# B&R Automation Studio project Task_1
Automation Studio 4.9

## Logical view

Binary libraries used (declarations not repeated): operator, runtime, astime, AsIecCon, Acp10man, Acp10par, NcGlobal, Acp10_MC, sys_lib, brsystem, Acp10sim, MpAxis, MpCom, MpBase, AsTCP, standard, AsArLog, AsBrStr

### Global.var - Global variables
```iecst
VAR RETAIN
	MyGlobal : {REDUND_UNREPLICABLE} UDINT := 10;
END_VAR
VAR
	gAxis01 : ACP10AXIS_typ;
	gAxis02 : ACP10AXIS_typ;
	START_BUTTON : BOOL;
	TRIGGER_INPUT : BOOL;
	EMERGENCY_STOP : BOOL;
	GreenLight : BOOL;
	RedLight : BOOL;
	CutterPosition : LREAL;
	ConveyorPosition : LREAL;
	STOP : BOOL;
	CONVEYOR_SPEED : {REDUND_UNREPLICABLE} INT := 0;
	EmergencyLight : BOOL;
	ERROR_RESET : BOOL;
	RealConveyorSpeed : INT;
	REG_TRIGGER : BOOL;
	CUTTER_POSITION : INT;
END_VAR
```

### Package Logical/Libraries - Global libraries

### Library Logical/Libraries/MyLib (IEC)

#### Types.typ - Exported data types
```iecst
TYPE
	GA_State :
		(
		NotPowered,
		WaitPower,
		Powered,
		CheckCommand,
		MoveVelocity,
		CheckVelocity,
		MoveAdditive,
		AxisHalt,
		AxisStop
		);
	COMMANDS :
		(
		NONE,
		MOVE_VELOCITY,
		MOVE_ADDITIVE,
		AXIS_HALT,
		AXIS_STOP
		);
END_TYPE
```

#### Constants.var - Exported constants
```iecst
VAR CONSTANT
	STANDSTILL : WORD := 2#00001000;
	DISCRETE_MOTION : WORD := 2#00010000;
	CONTINUOUS_MOTION : WORD := 2#00100000;
	CUTTER_SPEED : REAL := 200.0;
	CUTTER_END_POSE : REAL := 50.0;
	BELT_DISTANCE : REAL := 100.0;
END_VAR
```

#### MyLib.fun - Exported functions and function blocks
```iecst
FUNCTION_BLOCK GenericAxis_FB (*$GROUP=User,$CAT=User,$GROUPICON=User.png,$CATICON=User.png*)
	VAR_INPUT
		AxisOperation : INT;
		AxisCommand : COMMANDS;
		Master : UDINT;
		Slave : UDINT;
		CamTable : STRING[12];
		Position : REAL;
		Velocity : REAL;
		Acceleration : REAL;
		Deceleration : REAL;
		Jerk : REAL;
		Direction : USINT;
		ArraySize : INT;
		Scale : REAL;
		Offset : REAL;
		RatioNumerator : INT;
		RatioDenominator : INT;
	END_VAR
	VAR_OUTPUT
		CommandExecuted : BOOL;
		CommandAborted : BOOL;
		Error : BOOL;
		ErrorID : UINT;
		AxisErrorID : UINT;
		AxisErrorCount : UINT;
		AxisNotInitialized : BOOL;
		Status : WORD;
		ActualVelocity : REAL;
		ActualPosition : LREAL;
	END_VAR
	VAR_IN_OUT
		AxisEnable : BOOL;
	END_VAR
	VAR
		OldVelocity : REAL;
		MC_Power_GA : MC_Power;
		MC_Home_GA : MC_Home;
		MC_MoveVelocity_GA : MC_MoveVelocity;
		MC_MoveAdditive_GA : MC_MoveAdditive;
		MC_MoveAbsolute_GA : MC_MoveAbsolute;
		MC_ReadActualPosition_GA : MC_ReadActualPosition;
		MC_ReadActualVelocity_GA : MC_ReadActualVelocity;
		MC_ReadAxisError_GA : MC_ReadAxisError;
		MC_ReadStatus_GA : MC_ReadStatus;
		AxisState : GA_State;
		MC_Halt_GA : MC_Halt;
		MC_Stop_GA : MC_Stop;
	END_VAR
END_FUNCTION_BLOCK
```

#### GenericAxis_FB.st
```iecst
FUNCTION_BLOCK GenericAxis_FB
	CASE (AxisState) OF
		NotPowered:
			IF AxisEnable THEN
				MC_Power_GA.Enable := TRUE;
				AxisState := WaitPower;
			END_IF;
		WaitPower:
			IF MC_Power_GA.Status THEN
				MC_Home_GA.Execute := TRUE;
				AxisState := Powered;
			END_IF;
		Powered:
			IF MC_Home_GA.Done THEN
				MC_Home_GA.Execute := FALSE;
				AxisEnable := FALSE;
				CommandExecuted := TRUE;
				AxisState := CheckCommand; //ready state in the prof's slides
			END_IF
		// In this state you can implement several commands
		CheckCommand:
			IF AxisCommand = MOVE_VELOCITY THEN
				CommandExecuted := FALSE;
				MC_MoveVelocity_GA.Execute := TRUE;
				AxisState := MoveVelocity;
			END_IF

			IF AxisCommand = MOVE_ADDITIVE THEN
				CommandExecuted := FALSE;
				MC_MoveAdditive_GA.Execute := TRUE;
				AxisState := MoveAdditive;
			END_IF

			IF AxisCommand = AXIS_HALT THEN
				CommandExecuted := FALSE;
				MC_Halt_GA.Execute := TRUE;
				AxisState := AxisHalt;
			END_IF

			IF AxisCommand = AXIS_STOP THEN
				CommandExecuted := FALSE;
				MC_Stop_GA.Execute := TRUE;
				AxisState := AxisStop;
			END_IF

			(*IF AxisCommand = NONE THEN
				CommandExecuted := FALSE;
			END_IF*)

		// command states
		MoveVelocity:
			IF MC_MoveVelocity_GA.InVelocity THEN
				CommandExecuted := TRUE;
				MC_MoveVelocity_GA.Execute := FALSE;
				AxisState := CheckVelocity;
			END_IF
			IF (AxisCommand <> MOVE_VELOCITY) THEN
				CommandExecuted := FALSE;
				AxisState := CheckCommand;
			END_IF
		CheckVelocity:
			IF (Velocity <> OldVelocity) THEN
				OldVelocity := Velocity;
				MC_MoveVelocity_GA.Execute := TRUE;
				AxisState := MoveVelocity;
			END_IF
			IF (AxisCommand <> MOVE_VELOCITY) THEN
				CommandExecuted := FALSE;
				AxisState := CheckCommand;

			END_IF

		MoveAdditive:
			IF MC_MoveAdditive_GA.Done THEN
				MC_MoveAdditive_GA.Execute := FALSE;
				AxisCommand := NONE;
				AxisState := CheckCommand;
				CommandExecuted := TRUE;
			ELSIF (AxisCommand <> MOVE_ADDITIVE) THEN
				MC_MoveAdditive_GA.Execute := FALSE;
				CommandExecuted := FALSE;
				AxisState := CheckCommand;

			END_IF

			// In my implementation I used Halt to stop in Emergency conditions. IT IS NOT CORRECT
			// TO DO: Implement Halt in normal conditions and use STOP for critical conditions
		AxisHalt:
			IF MC_Halt_GA.Done THEN
				CommandExecuted := TRUE;
				MC_Halt_GA.Execute := FALSE;
				AxisState := NotPowered; // It goes to the NotPowered state to perform a full reset of the system
				MC_Power_GA.Enable := FALSE; // The power is disabled for the same reason
				AxisCommand := NONE;
			END_IF

		// TO DO: IT IS NOT IMPLEMENTED  (To stop the execution in critical conditions)
		AxisStop:
			IF MC_Stop_GA.Done THEN
				CommandExecuted := TRUE;
				MC_Stop_GA.Execute := FALSE;
				AxisState := NotPowered; // It goes to the NotPowered state to perform a full reset of the system
				MC_Power_GA.Enable := FALSE; // The power is disabled for the same reason
				AxisCommand := NONE;
			END_IF
	END_CASE;

	MC_Power_GA.Axis := Slave;
	MC_Power_GA();
	MC_Home_GA.Axis := Slave;
	MC_Home_GA.Position := 0;
	MC_Home_GA();
	MC_MoveVelocity_GA.Axis := Slave;
	MC_MoveVelocity_GA.Velocity := Velocity;
	MC_MoveVelocity_GA.Acceleration := Acceleration;
	MC_MoveVelocity_GA.Deceleration := Deceleration;
	MC_MoveVelocity_GA();

	MC_MoveAdditive_GA.Axis := Slave;
	MC_MoveAdditive_GA.Distance := Position;
	MC_MoveAdditive_GA.Velocity := Velocity;
	MC_MoveAdditive_GA.Acceleration := Acceleration;
	MC_MoveAdditive_GA.Deceleration := Deceleration;
	MC_MoveAdditive_GA();

	// Stop in normal conditions
	MC_Halt_GA.Axis := Slave;
	MC_Halt_GA.Deceleration := Deceleration;
	MC_Halt_GA();

	// Stop in critical conditions
	MC_Stop_GA.Axis := Slave;
	MC_Stop_GA.Deceleration := Deceleration;
	MC_Stop_GA();

	// FEEDBACKS
	MC_ReadActualPosition_GA.Axis := Slave;
	MC_ReadActualPosition_GA.Enable := TRUE;
	MC_ReadActualPosition_GA();
	ActualPosition := MC_ReadActualPosition_GA.Position;
	MC_ReadActualVelocity_GA.Axis := Slave;
	MC_ReadActualVelocity_GA.Enable := TRUE;
	MC_ReadActualVelocity_GA();
	ActualVelocity := MC_ReadActualVelocity_GA.Velocity;
	MC_ReadAxisError_GA.Enable := TRUE;
	MC_ReadAxisError_GA.Axis := Slave;
	MC_ReadAxisError_GA();
	Error := MC_ReadAxisError_GA.Error;
	ErrorID := MC_ReadAxisError_GA.ErrorID;
	AxisErrorID := MC_ReadAxisError_GA.AxisErrorID;
	AxisErrorCount := MC_ReadAxisError_GA.AxisErrorCount;
	MC_ReadStatus_GA.Enable := TRUE;
	MC_ReadStatus_GA.Axis := Slave;
	MC_ReadStatus_GA();

	IF MC_ReadStatus_GA.ContinuousMotion THEN
		Status := CONTINUOUS_MOTION;
	END_IF
	IF MC_ReadStatus_GA.DiscreteMotion THEN
		Status := DISCRETE_MOTION;
	END_IF
	IF MC_ReadStatus_GA.StandStill THEN
		Status := STANDSTILL;
	END_IF
END_FUNCTION_BLOCK
```

### Library Logical/Libraries/ComTCP/ComTCP_L (ANSIC)

#### MNG_CpyMsgToInp.cpp
```cpp
#include "MNG_InternalTyp.hpp"

unsigned long int MNG_CpyMsgToInp(MNG_RawDatagram * pFromServer, ComTCP_INPUTS_32BIT_FWRD *pSimInputs) {

    MNG_DatagramType datagramType;
	unsigned long int DWordBuffer;
        unsigned long int byteCount;
	unsigned long int numSignalsInMessage;

	byteCount = N_TO_HUDINT((pFromServer->Header).ByteCount);
	datagramType = static_cast<MNG_DatagramType>(N_TO_HUDINT((pFromServer->Header).DatagramType));
	if (datagramType != MNG_Raw32BitImage) {
		return 0;
	}

    pSimInputs->NumSignals = 15;

    numSignalsInMessage = N_TO_HUDINT(pFromServer->Payload[0]);
        if ((static_cast<long int>(numSignalsInMessage) != pSimInputs->NumSignals) ||
	(byteCount != 4 + numSignalsInMessage * 4)) {
		return 0;
	}

    /* BOOL Emergency_Button_ButtonToggle */
    pSimInputs->Emergency_Button_ButtonToggle = (pFromServer->Payload[1] != 0);

    /* BOOL Yellow_Button_ButtonPress */
    pSimInputs->Yellow_Button_ButtonPress = (pFromServer->Payload[2] != 0);

    /* BOOL White_Button_ButtonPress */
    pSimInputs->White_Button_ButtonPress = (pFromServer->Payload[3] != 0);

    /* BOOL Start_Button_ButtonPress */
    pSimInputs->Start_Button_ButtonPress = (pFromServer->Payload[4] != 0);

    /* BOOL Stop_Button_ButtonPress */
    pSimInputs->Stop_Button_ButtonPress = (pFromServer->Payload[5] != 0);

    /* FLOAT32 Knob_0_AXIS */
    DWordBuffer = N_TO_HUDINT(pFromServer->Payload[6]);
    brsmemcpy((unsigned long int)&(pSimInputs->Knob_0_AXIS), (unsigned long int)&(DWordBuffer), 4);

    /* FLOAT32 Knob_1_AXIS */
    DWordBuffer = N_TO_HUDINT(pFromServer->Payload[7]);
    brsmemcpy((unsigned long int)&(pSimInputs->Knob_1_AXIS), (unsigned long int)&(DWordBuffer), 4);

    /* FLOAT32 Knob_2_AXIS */
    DWordBuffer = N_TO_HUDINT(pFromServer->Payload[8]);
    brsmemcpy((unsigned long int)&(pSimInputs->Knob_2_AXIS), (unsigned long int)&(DWordBuffer), 4);

    /* FLOAT32 Knob_3_AXIS */
    DWordBuffer = N_TO_HUDINT(pFromServer->Payload[9]);
    brsmemcpy((unsigned long int)&(pSimInputs->Knob_3_AXIS), (unsigned long int)&(DWordBuffer), 4);

    /* FLOAT32 Shaft_1_AXIS */
    DWordBuffer = N_TO_HUDINT(pFromServer->Payload[10]);
    brsmemcpy((unsigned long int)&(pSimInputs->Shaft_1_AXIS), (unsigned long int)&(DWordBuffer), 4);

    /* BOOL Shaft_1_LBK */
    pSimInputs->Shaft_1_LBK = (pFromServer->Payload[11] != 0);

    /* BOOL Shaft_1_LFR */
    pSimInputs->Shaft_1_LFR = (pFromServer->Payload[12] != 0);

    /* FLOAT32 Shaft_0_AXIS */
    DWordBuffer = N_TO_HUDINT(pFromServer->Payload[13]);
    brsmemcpy((unsigned long int)&(pSimInputs->Shaft_0_AXIS), (unsigned long int)&(DWordBuffer), 4);

    /* BOOL Shaft_0_LBK */
    pSimInputs->Shaft_0_LBK = (pFromServer->Payload[14] != 0);

    /* BOOL Shaft_0_LFR */
    pSimInputs->Shaft_0_LFR = (pFromServer->Payload[15] != 0);

return N_TO_HUDINT((pFromServer->Header).Counter); // return counter
}
```

#### MNG_CpyOutToMsg.cpp
```cpp
#include "MNG_InternalTyp.hpp"

unsigned long int MNG_CpyOutToMsg(MNG_RawDatagram * pToServer, unsigned long int counter, ComTCP_OUTPUTS_32BIT_FWRD *pSimOutputs ) {

        unsigned long int DWordBuffer;

        pSimOutputs->NumSignals = 6;
        (pToServer->Header).ByteCount    = H_TO_NUDINT(28);
        (pToServer->Header).DatagramType = H_TO_NUDINT(MNG_Raw32BitImage);
        (pToServer->Header).SentTime = H_TO_NUDINT(0);  // Todo
        (pToServer->Header).Counter = H_TO_NUDINT(counter);
        pToServer->Payload[0] = H_TO_NUDINT(pSimOutputs->NumSignals);

    /* Yellow_light_Key : UINT32 */
    pToServer->Payload[1] = H_TO_NUDINT(pSimOutputs->Yellow_light_Key);

    /* Stop_light_Key : UINT32 */
    pToServer->Payload[2] = H_TO_NUDINT(pSimOutputs->Stop_light_Key);

    /* White_light_Key : UINT32 */
    pToServer->Payload[3] = H_TO_NUDINT(pSimOutputs->White_light_Key);

    /* Green_light_Key : UINT32 */
    pToServer->Payload[4] = H_TO_NUDINT(pSimOutputs->Green_light_Key);

    /* Shaft_0_ACT_POS : FLOAT32 */
    brsmemcpy((unsigned long int)&(DWordBuffer), (unsigned long int)&(pSimOutputs->Shaft_0_ACT_POS), 4);
    pToServer->Payload[5] = H_TO_NUDINT(DWordBuffer);

    /* Shaft_1_ACT_POS : FLOAT32 */
    brsmemcpy((unsigned long int)&(DWordBuffer), (unsigned long int)&(pSimOutputs->Shaft_1_ACT_POS), 4);
    pToServer->Payload[6] = H_TO_NUDINT(DWordBuffer);

	return 0;
}
```

### Package Logical/gAxis01obj - gAxis01obj

### gAxis01i.ax
```
InitParameter (Version=5.24.1, NcSwId=ACP10)
  ACP10AXIS_typ:
    dig_in:
      level:
        reference = ncACTIV_HI
        pos_hw_end = ncACTIV_HI
        neg_hw_end = ncACTIV_HI
        trigger1 = ncACTIV_HI
        trigger2 = ncACTIV_HI
    encoder_if:
      parameter:
        count_dir = ncSTANDARD
        scaling:
          load:
            units = 360
            rev_motor = 1
    limit:
      parameter:
        v_pos = 10000.0
        v_neg = 10000.0
        a1_pos = 50000.0
        a2_pos = 50000.0
        a1_neg = 50000.0
        a2_neg = 50000.0
        t_jolt = 0.0
        t_in_pos = 0.0
        pos_sw_end = 2000000000
        neg_sw_end = -2000000000
        ds_warning = 500.0
        ds_stop = 1000.0
        a_stop = 1.0E+30
        dv_stop = 0.0
        dv_stop_mode = ncOFF
    controller:
      mode = ncPOSITION
      position:
        kv = 349.0
        tn = 0.0
        t_predict = 0.0004
        t_total = 0.0004
        p_max = 1.0E+30
        i_max = 0.0
      speed:
        kv = 0.65
        tn = 0.0
        t_filter = 0.0
        isq_filter1:
          type = ncOFF
          a0 = 0.0
          a1 = 0.0
          b0 = 0.0
          b1 = 0.0
          b2 = 0.0
          c0_par_id = 0
          c1_par_id = 0
        isq_filter2:
          type = ncOFF
          a0 = 0.0
          a1 = 0.0
          b0 = 0.0
          b1 = 0.0
          b2 = 0.0
          c0_par_id = 0
          c1_par_id = 0
        isq_filter3:
          type = ncOFF
          a0 = 0.0
          a1 = 0.0
          b0 = 0.0
          b1 = 0.0
          b2 = 0.0
          c0_par_id = 0
          c1_par_id = 0
      uf:
        type = ncLINEAR + ncCORRECTION
        auto_config = ncMOTOR_PAR
        u0 = 0.0
        un = 0.0
        fn = 50.0
        k_f_slip = 0.0
      ff:
        mode = ncSTANDARD
        torque_load = 0.0
        torque_pos = 0.0
        torque_neg = 0.0
        kv_torque = 0.0
        inertia = 0.0
        t_filter_a = 0.0
      fb:
        mode = ncSTANDARD
        speed_mix_ratio = 0.0
        speed_kv = 0.0
      model:
        mass1:
          inertia = 0.0
          viscous_friction = 0.0
        mass2:
          inertia = 0.0
          viscous_friction = 0.0
          stiffness = 0.0
          damping = 0.0
    move:
      stop:
        parameter[0]:
          decel_ramp = ncA_LIMIT
          controller = ncON
        parameter[1]:
          decel_ramp = ncA_LIMIT
          controller = ncON
        parameter[2]:
          decel_ramp = ncA_LIMIT
          controller = ncON
        parameter[3]:
          decel_ramp = ncA_LIMIT
          controller = ncON
        quickstop:
          decel_ramp = ncA_LIMIT
          t_jolt = 0.0
        drive_error:
          decel_ramp = ncA_LIMIT
      homing:
        parameter:
          s = 0
          v_switch = 5000.0
          v_trigger = 500.0
          a = 50000.0
          mode = ncDIRECT
          edge_sw = ncPOSITIVE
          start_dir = ncPOSITIVE
          trigg_dir = ncPOSITIVE
          ref_pulse = ncOFF
          fix_dir = ncOFF
          tr_s_block = 0.0
          torque_lim = 0.0
          ds_block = 0.0
          ds_stop = 0.0
      basis:
        parameter:
          v_pos = 360.0
          v_neg = 5000.0
          a1_pos = 50000.0
          a2_pos = 50000.0
          a1_neg = 50000.0
          a2_neg = 50000.0
    message:
      text:
        parameter:
          format = ncBREAK
          columns = 80
          data_modul = acp10etxen
```

### Program Logical/PROGRAM1 (IEC)

#### Types.typ
```iecst
TYPE
	State_type :
		(
		CutterMoveBackward,
		CutterCompleted,
		CutterMoveForward,
		ConveyorStopping,
		ConveyorMoving,
		ConveyorStarting,
		AxisEnabled,
		InitializeAxis,
		CutterBackward,
		CutterForward,
		ConveyorHolding,
		WaitProduct,
		Initialize,
		Init,
		StopState,
		HaltState,
		WaitForConveyor,
		CheckReset,
		RegulatePosition
		);
END_TYPE
```

#### Variables.var
```iecst
VAR
	MachineState : State_type;
	ConveyorEnable : BOOL;
	CutterEnable : BOOL;
	Cutter : GenericAxis_FB;
	Conveyor : GenericAxis_FB;
	InitializeConveyor : BOOL;
	InitializeCutter : BOOL;
	ConveyorDisable : BOOL;
	CutterDisable : BOOL;
	ConveyorState : State_type;
	CutterState : State_type;
	ConveyorAxisEnable : BOOL;
	CutterAxisEnable : BOOL;
	FutureStop : BOOL;
	CoveyorState : BOOL;
	ConveyorStopped : BOOL;
	CutterStopped : BOOL;
	EmergencyStateMachine : INT;
	Count : INT;
	ToggleLights : BOOL;
	OldCutterPose : INT;
END_VAR
```

#### Main.st
```iecst
PROGRAM _INIT
	(* Insert code here *)
	MachineState := Init;
	ConveyorState := Init;
	CutterState := Init;
	OldCutterPose := 0;
END_PROGRAM

PROGRAM _CYCLIC

	// STOP indicates an emergency stop, it is not a stop in normal conditions
	CASE EmergencyStateMachine OF
		0 :
			IF EMERGENCY_STOP THEN
				MachineState := StopState;
				ConveyorState := StopState;
				CutterState := StopState;
				Conveyor.AxisCommand := AXIS_HALT;
				Cutter.AxisCommand := AXIS_HALT;
				EmergencyStateMachine := 1;
			END_IF
		1 :
			IF NOT EMERGENCY_STOP AND CutterStopped AND ConveyorStopped THEN
				EmergencyStateMachine := 0;
			END_IF
	END_CASE

	IF STOP THEN
		FutureStop := TRUE;
	END_IF

	// GLOBAL STATE MACHINE
	CASE MachineState OF
		Init: // Initial configuration state
			IF START_BUTTON THEN
				InitializeConveyor := TRUE;
				InitializeCutter := TRUE;
				MachineState := Initialize;
			END_IF
		Initialize: // initialization - Power and Homing (This operations are implemented inside the function block)
			IF NOT InitializeConveyor AND NOT InitializeCutter THEN
				ConveyorEnable := TRUE;
				MachineState := WaitProduct;
			END_IF
		WaitProduct: // It waits for a trigger
			IF NOT ConveyorEnable AND TRIGGER_INPUT AND NOT REG_TRIGGER THEN
				ConveyorDisable := TRUE;
				MachineState := ConveyorHolding;
			END_IF
			// STOP
			IF FutureStop THEN
				MachineState := HaltState;
			END_IF

		ConveyorHolding: // Stop the Conveyor
			IF NOT ConveyorDisable THEN
				CutterEnable := TRUE;
				MachineState := CutterForward;
			END_IF
		CutterForward: // Cut
			IF NOT CutterEnable THEN
				CutterDisable := TRUE;
				MachineState := CutterBackward;
			END_IF
		CutterBackward: // Go back
			IF NOT CutterDisable THEN
				ConveyorEnable := TRUE;
				MachineState := WaitProduct;
			END_IF

		// Emergency stop
		StopState:
			IF NOT EMERGENCY_STOP AND ConveyorStopped AND CutterStopped THEN
				MachineState := CheckReset;
			END_IF
		CheckReset:
			IF ERROR_RESET THEN
				MachineState := Init;
				ConveyorStopped := FALSE;
				CutterStopped := FALSE;
				FutureStop := FALSE;
			END_IF
		// CAN BE ERASED
		HaltState:
			IF ConveyorStopped AND CutterStopped THEN
				MachineState := Init;
				ConveyorStopped := FALSE;
				CutterStopped := FALSE;
				FutureStop := FALSE;
			END_IF

	END_CASE

	// CONVEYOR STATE MACHINE
	CASE ConveyorState OF
		Init:
			IF InitializeConveyor THEN
				ConveyorAxisEnable := TRUE;
				ConveyorState := InitializeAxis;
			END_IF
		InitializeAxis:
			IF NOT ConveyorAxisEnable THEN
				InitializeConveyor := FALSE;
				ConveyorState := AxisEnabled;
			END_IF
		AxisEnabled:
			IF ConveyorEnable AND NOT FutureStop THEN
				Conveyor.AxisCommand := MOVE_VELOCITY;
				ConveyorState := ConveyorStarting;
			ELSIF FutureStop THEN
				Conveyor.AxisCommand := AXIS_HALT;
				ConveyorState := HaltState;
			END_IF
		ConveyorStarting:
			IF Conveyor.CommandExecuted THEN
				ConveyorEnable := FALSE;
				ConveyorState := ConveyorMoving;
			END_IF
		ConveyorMoving:
			IF ConveyorDisable AND NOT FutureStop THEN
				Conveyor.AxisCommand := MOVE_ADDITIVE;
				ConveyorState := ConveyorStopping;
			ELSIF FutureStop THEN
				Conveyor.AxisCommand := AXIS_HALT;
				ConveyorState := HaltState;
			END_IF
		ConveyorStopping:
			IF Conveyor.CommandExecuted THEN
				ConveyorDisable := FALSE;
				ConveyorState := AxisEnabled;
			END_IF

		// EMERGENCY STOP
		StopState:
			IF NOT EMERGENCY_STOP AND Conveyor.CommandExecuted THEN
				ConveyorEnable := FALSE;
				ConveyorDisable := FALSE;
				ConveyorStopped := TRUE;
				ConveyorState := Init;
			END_IF

		HaltState:
			IF Conveyor.CommandExecuted THEN
				ConveyorDisable := FALSE;
				ConveyorEnable := FALSE;
				ConveyorStopped := TRUE;
				ConveyorState := Init;
			END_IF
	END_CASE

	// CUTTER STATE MACHINE
	CASE CutterState OF
		Init:
			IF InitializeCutter THEN
				CutterAxisEnable := TRUE;
				CutterState := InitializeAxis;
			END_IF
		InitializeAxis:
			IF NOT CutterAxisEnable THEN
				InitializeCutter := FALSE;
				CutterState := AxisEnabled;
			END_IF
		AxisEnabled:
			IF REG_TRIGGER THEN // 2
				IF CUTTER_POSITION <> OldCutterPose THEN
					Cutter.Position := INT_TO_REAL((CUTTER_POSITION - OldCutterPose) / 100);
					OldCutterPose := CUTTER_POSITION;
					Cutter.AxisCommand := MOVE_ADDITIVE;
					CutterState := RegulatePosition;
				END_IF
			ELSIF ConveyorDisable AND NOT FutureStop THEN
				CutterState := WaitForConveyor;
			ELSIF FutureStop THEN
				Cutter.AxisCommand := AXIS_HALT;
				CutterState := HaltState;
			END_IF

		RegulatePosition: // 2
			IF Cutter.CommandExecuted THEN
				CutterState := AxisEnabled;
			END_IF

		WaitForConveyor:
			IF CutterEnable THEN
				Cutter.Position := BELT_DISTANCE; // Added by me
				Cutter.AxisCommand := MOVE_ADDITIVE;
				CutterState := CutterMoveForward;
			END_IF
		CutterMoveForward:
			IF Cutter.CommandExecuted THEN
				CutterEnable := FALSE;
				CutterState := CutterCompleted;
			END_IF
		CutterCompleted:
			IF CutterDisable THEN
				Cutter.Position := -BELT_DISTANCE; // Added by me
				Cutter.AxisCommand := MOVE_ADDITIVE;
				CutterState := CutterMoveBackward;
			END_IF
		CutterMoveBackward:
			IF Cutter.CommandExecuted THEN
				CutterDisable := FALSE;
				CutterState := AxisEnabled;
			END_IF

		// EMERGENCY STOP
		StopState:
			IF NOT EMERGENCY_STOP AND Cutter.CommandExecuted THEN
				CutterEnable := FALSE;
				CutterDisable := FALSE;
				CutterStopped := TRUE;
				CutterState := Init;
			END_IF

		HaltState:
			IF Cutter.CommandExecuted THEN
				CutterDisable := FALSE;
				CutterEnable := FALSE;
				CutterStopped := TRUE;
				CutterState := Init;
			END_IF
	END_CASE

	// Counter for blink
	Count := Count + 1;
	IF Count = 10 THEN
		ToggleLights := TRUE;
		Count := 0;
	ELSE
		ToggleLights := FALSE;
	END_IF

	// LIGHTS
	IF MachineState = Init THEN
		IF ToggleLights THEN
			GreenLight := NOT GreenLight;
		END_IF
		RedLight := FALSE;
		EmergencyLight := FALSE;

	ELSIF MachineState <> HaltState AND MachineState <> StopState AND MachineState <> CheckReset THEN
		GreenLight := TRUE;
		RedLight := TRUE;
		EmergencyLight := FALSE;
	ELSIF MachineState = StopState OR MachineState = CheckReset THEN
		GreenLight := FALSE;
		RedLight := FALSE;
		IF ToggleLights THEN
			EmergencyLight := NOT EmergencyLight;
		END_IF
	END_IF

	Conveyor.Slave := ADR(gAxis01);
	Conveyor.Position := 2*BELT_DISTANCE;
	RealConveyorSpeed := CONVEYOR_SPEED/10;

	Conveyor.Velocity :=  INT_TO_REAL(RealConveyorSpeed);
	Conveyor.Acceleration := 200;
	Conveyor.Deceleration := 200;

	Conveyor(AxisEnable := ConveyorAxisEnable);
	ConveyorPosition := Conveyor.ActualPosition;

	Cutter.Slave := ADR(gAxis02);
	Cutter.Velocity := CUTTER_SPEED;
	Cutter.Acceleration := 200;
	Cutter.Deceleration := 200;

	Cutter(AxisEnable := CutterAxisEnable);
	CutterPosition := Cutter.ActualPosition;

END_PROGRAM

PROGRAM _EXIT
	(* Insert code here *)

END_PROGRAM
```

### MNG_Package.var
```iecst
(*                                                                            *)
(* File generated by the B&R AS 4 control config generator                    *)
(*                                                                            *)
(*     Provider: machineering                                                 *)
(*  Application: industrialPhysics_2.4.master                                 *)
(* Architecture: Windows 64 Bit                                               *)
(*      Version: 2.4.10491.master                                             *)
(*        Build: 164f85bec                                                    *)
(*         Date: 2020-03-30, Time: 13:49:25                                   *)
(*                                                                            *)

                VAR
                ComTCP_SimInputs : ComTCP_INPUTS_32BIT := (0);
    ComTCP_SimOutputs : ComTCP_OUTPUTS_32BIT := (0);

    ComTCP_SimServerAddress : STRING[15] := '127.0.0.1';
    ComTCP_SimServerPort : UINT := 5000;
    ComTCP_SimSendCycleTime : TIME := T#10ms;
    ComTCP_SimActive : BOOL := FALSE;

                END_VAR
```

### Program Logical/OutputBridge (IEC)

#### Main.st
```iecst
PROGRAM _INIT
	(* Insert code here *)

END_PROGRAM

PROGRAM _CYCLIC
	(* Insert code here *)
	ComTCP_SimOutputs.Green_light_Key := GreenLight;
	ComTCP_SimOutputs.Stop_light_Key := RedLight;
	ComTCP_SimOutputs.Yellow_light_Key := EmergencyLight;
	ComTCP_SimOutputs.Shaft_0_ACT_POS := LREAL_TO_REAL(ConveyorPosition);
	ComTCP_SimOutputs.Shaft_1_ACT_POS := LREAL_TO_REAL(CutterPosition);

END_PROGRAM

PROGRAM _EXIT
	(* Insert code here *)

END_PROGRAM
```

### Program Logical/InputBridge (IEC)

#### Main.st
```iecst
PROGRAM _INIT
	(* Insert code here *)

END_PROGRAM

PROGRAM _CYCLIC
	(* Insert code here *)
	START_BUTTON := ComTCP_SimInputs.Start_Button_ButtonPress;
	TRIGGER_INPUT := ComTCP_SimInputs.White_Button_ButtonPress;
	EMERGENCY_STOP := ComTCP_SimInputs.Emergency_Button_ButtonToggle;
	STOP := ComTCP_SimInputs.Stop_Button_ButtonPress;
	ERROR_RESET := ComTCP_SimInputs.Yellow_Button_ButtonPress;

END_PROGRAM

PROGRAM _EXIT
	(* Insert code here *)

END_PROGRAM
```

### Variables.var
```iecst
VAR
	State : State_type;
	GA_test : GenericAxis_FB;
	velocity : REAL := 100;
	ConveyorEnable : BOOL;
	CutterEnable : BOOL;
	Enable : BOOL;
	result : INT;
	Command : WORD := MOVE_VELOCITY;
	Actuation : INT;
	Cutter : GenericAxis_FB;
	Conveyor : GenericAxis_FB;
END_VAR
```

Listed in the project but not available here: Logical/Global.typ, Logical/Libraries/ComTCP/ComTCP_P, Logical/acp10etxen, Logical/gAxis02obj, Logical/MNG_Package.typ, Logical/MNG_Global.typ
